Fanuc KAREL source: kb00094.KL

-- PROVISIONAL review KL for V940-1; original PC SHA256 7ea418669fc3570ab6ccebc37dd5b6fb7ec4b78d9eeffcb69544e3396d65d2de
-- Incomplete behavior may be omitted. Consult companion uncertainty JSON. Do not deploy.
PROGRAM KB00094
%NOLOCKGROUP
BEGIN
  -- V9_ZERO_TABLE_METADATA_HINT layout=0002_ascii; no indexed target words; source/name/runtime held
  -- UNRESOLVED_PC offsets 5-12; opcodes 9D,23
  -- UNRESOLVED_PC offsets 17-27; opcodes 27,22,31
  -- UNRESOLVED_PC offsets 32-36; opcodes 7F
END KB00094
